Staubli VAL3: toPointRxMillis.pgx

public program toPointRxMillis(num& x_nPositionArray[], pointRx& x_pPointRx)
  local num l_nScaleFactor
begin
  l_nScaleFactor = 1000.0
  x_pPointRx.trsf.x = x_nPositionArray[0] * l_nScaleFactor
  x_pPointRx.trsf.y = x_nPositionArray[1] * l_nScaleFactor
  x_pPointRx.trsf.z = x_nPositionArray[2] * l_nScaleFactor
end
